PROGRAM SLOW
VAR
END_VAR

;

END_PROGRAM

(* stored: Version 1.1.0.1, ProductVersion 3.1.4024.9
   POU SLOW: Id {3bd6c98f-32d6-4aaa-ac41-823b5a11695e}, SpecialFunc None *)
